// SIMATIC STEP 7 (V5.x) project Lit_servis
// CPU: CPU 312
// station: Hardware
// station: SIMATIC 300(1)
// station: P_ADR_BUS
// station: P_ADR_BUS
// station: Configuration
// program: S7 Program(6)

SYMBOL_TABLE
"s3.1-3.3"	I 4.0	BOOL	// авар. откл.ГП
"s3.4"	I 4.1	BOOL	// откл. вентилятора.
"s3.5"	I 4.2	BOOL	// вкл. вентилятора
"s3.6"	I 4.3	BOOL	// нормальное откл.ГП
"s3.7"	I 4.4	BOOL	// вкл. ГП
"s4.1"	I 4.5	BOOL	// выбор режима
"s4.2"	I 4.6	BOOL	// не используется в ПрП
"s4.3"	I 4.7	BOOL	// не используется в ПрП
"s1.1-1.2"	I 5.0	BOOL	// конеч. пол. левого 1
"s1.3-1.4"	I 5.1	BOOL	// конеч. пол. правого 1
"s1.5-1.6"	I 5.2	BOOL	// конеч. пол. левого 2
"s1.7-1.8"	I 5.3	BOOL	// конеч. пол. правого 2
"s1.9-1.10"	I 5.4	BOOL	// поднятие магазина
"s1.11"	I 5.5	BOOL	// положение штурвала
"s1.12"	I 5.6	BOOL	// контроль вентилятора
"B1.1"	I 5.7	BOOL	// наличие воздуха
"F1.1-1.3"	I 6.0	BOOL	// тепловое реле
"B8.1"	I 6.1	BOOL	// наличие крышки-левая
"B8.2"	I 6.2	BOOL	// сектор-левая
"B8.3"	I 6.3	BOOL	// наличие крышки-правая
"B8.4"	I 6.4	BOOL	// сектор-правая
"B8.5"	I 6.5	BOOL	// счётчик-левая
"B8.6"	I 6.6	BOOL	// счётчик-правая
"B8.7"	I 6.7	BOOL	// мёртвая точка
"B8.9"	I 7.0	BOOL	// min. магазин 1-левый
"B8.10"	I 7.1	BOOL	// max. магазин 1-левый
"B8.11"	I 7.2	BOOL	// min. магазин 2-правый
"B8.12"	I 7.3	BOOL	// max. магазин 2-правый
"K9.1"	Q 10.0	BOOL	// управление вентилятором
"K9.3"	Q 10.1	BOOL	// управление осн. нагревателем
"K9.4"	Q 10.2	BOOL	// управление 1 доп.. нагревателем
"K9.5"	Q 10.3	BOOL	// управление 2 доп.. нагревателем
"K9.6"	Q 10.4	BOOL	// управление-маг. колесо
"K9.7"	Q 10.5	BOOL	// управление-привод гумир.
"K1.12"	Q 10.6	BOOL	// управление-привод ГП
"K7.5"	Q 11.0	BOOL	// управление подачей крышек-магазин 1(левый)
"K7.10"	Q 11.1	BOOL	// управление подачей крышек-магазин 2(правый)
"K7.6"	Q 11.2	BOOL	// управление-грибок магазин 1(левый)
"K7.11"	Q 11.3	BOOL	// управление-грибок магазин 2(правый)
"Y2.1"	Q 11.4	BOOL	// подача пасты-левый
"Y2.2"	Q 11.5	BOOL	// подача пасты-правый
"Y2.9"	Q 11.6	BOOL	// управление тормозом
"VAT_1"	VAT 1	
END_SYMBOL_TABLE

FUNCTION FC 1 : VOID
VERSION : 0.1
BEGIN
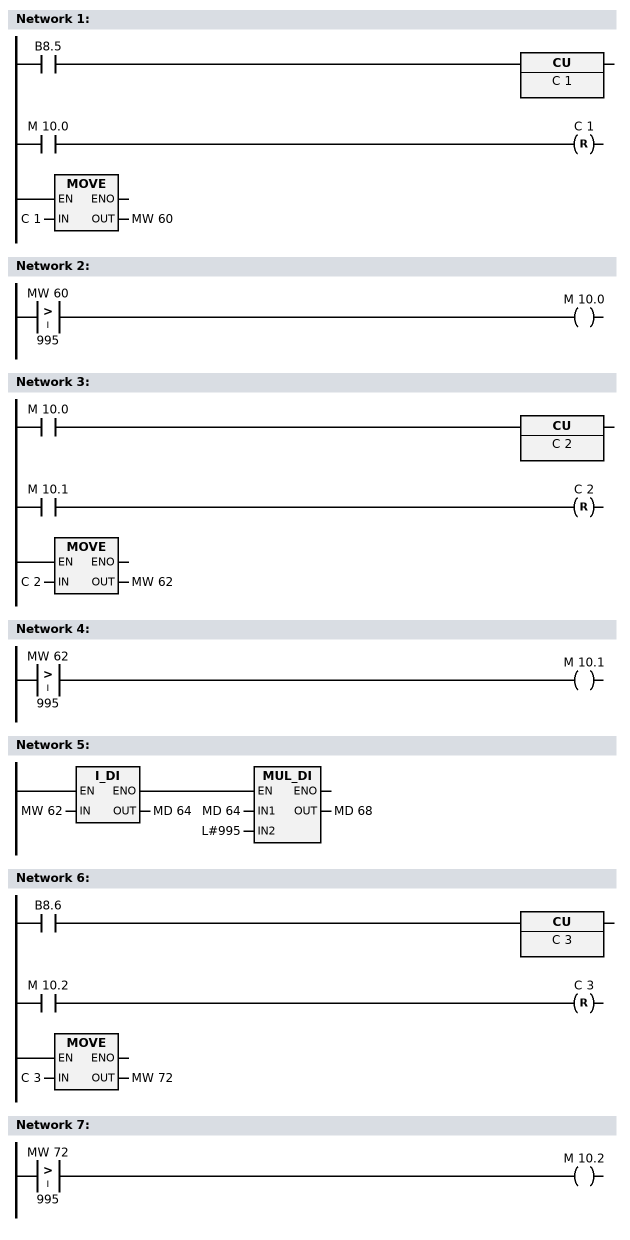
NETWORK
TITLE =
      A     "B8.5";
      CU    C 1;
      BLD   101;
      NOP   0;
      NOP   0;
      A     M 10.0;
      R     C 1;
      L     C 1;
      T     MW 60;
      NOP   0;
      NOP   0;
NETWORK
TITLE =
      L     MW 60;
      L     995;
      >I;
      =     M 10.0;
NETWORK
TITLE =
      A     M 10.0;
      CU    C 2;
      BLD   101;
      NOP   0;
      NOP   0;
      A     M 10.1;
      R     C 2;
      L     C 2;
      T     MW 62;
      NOP   0;
      NOP   0;
NETWORK
TITLE =
      L     MW 62;
      L     995;
      >I;
      =     M 10.1;
NETWORK
TITLE =
      A(;
      L     MW 62;
      ITD;
      T     MD 64;
      SET;
      SAVE;
      CLR;
      A     BR;
      );
      JNB   _001;
      L     MD 64;
      L     L#995;
      *D;
      T     MD 68;
_001: NOP   0;
NETWORK
TITLE =
      A     "B8.6";
      CU    C 3;
      BLD   101;
      NOP   0;
      NOP   0;
      A     M 10.2;
      R     C 3;
      L     C 3;
      T     MW 72;
      NOP   0;
      NOP   0;
NETWORK
TITLE =
      L     MW 72;
      L     995;
      >I;
      =     M 10.2;
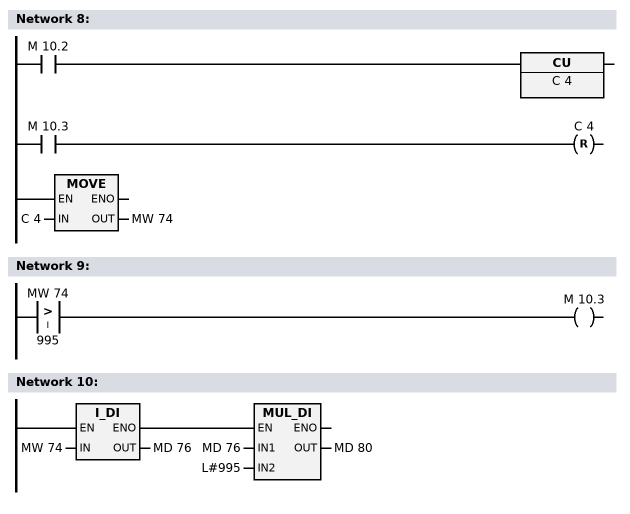
NETWORK
TITLE =
      A     M 10.2;
      CU    C 4;
      BLD   101;
      NOP   0;
      NOP   0;
      A     M 10.3;
      R     C 4;
      L     C 4;
      T     MW 74;
      NOP   0;
      NOP   0;
NETWORK
TITLE =
      L     MW 74;
      L     995;
      >I;
      =     M 10.3;
NETWORK
TITLE =
      A(;
      L     MW 74;
      ITD;
      T     MD 76;
      SET;
      SAVE;
      CLR;
      A     BR;
      );
      JNB   _002;
      L     MD 76;
      L     L#995;
      *D;
      T     MD 80;
_002: NOP   0;
NETWORK
TITLE =
END_FUNCTION

FUNCTION FC 2 : VOID
//Счётчики
VERSION : 0.1
BEGIN
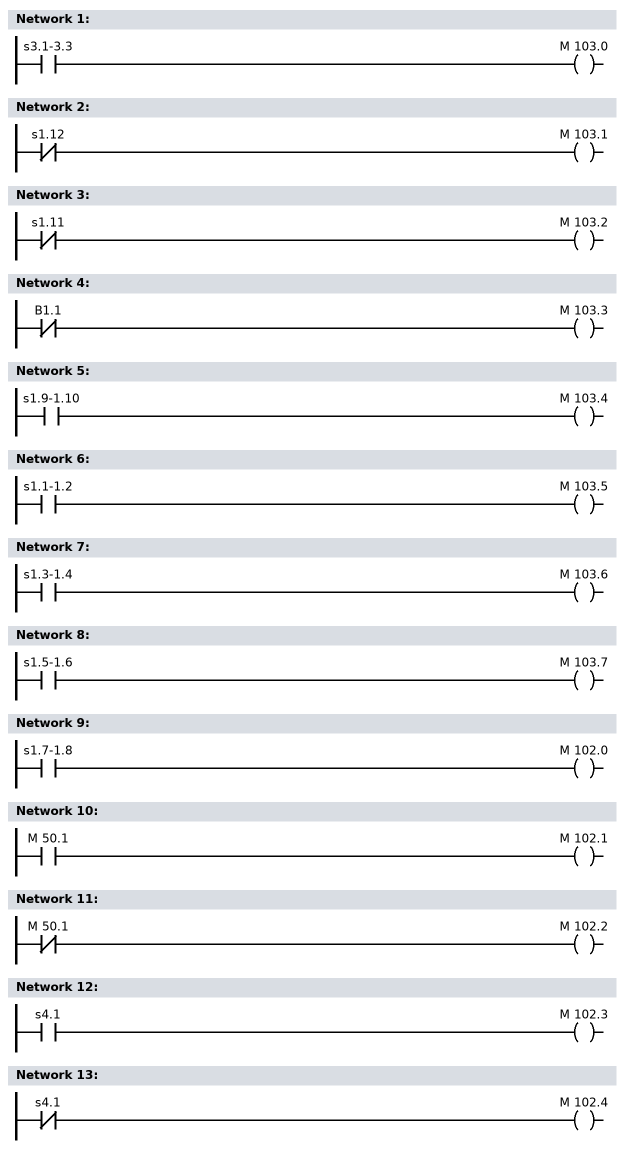
NETWORK
TITLE =
//Сообщение:аврийное отключение ГП
      A     "s3.1-3.3";
      =     M 103.0;
NETWORK
TITLE =
//Сообщение:вентилятор отключился
      AN    "s1.12";
      =     M 103.1;
NETWORK
TITLE =
//Сообщение:штурвал не в "автомате"
      AN    "s1.11";
      =     M 103.2;
NETWORK
TITLE =
//Сообщение:отсутствует воздух в системе
      AN    "B1.1";
      =     M 103.3;
NETWORK
TITLE =
//Сообщение:гумировочная головка магазин крышек подняты
      A     "s1.9-1.10";
      =     M 103.4;
NETWORK
TITLE =
//Сообщение:конечное положение левого 1 шнека
      A     "s1.1-1.2";
      =     M 103.5;
NETWORK
TITLE =
//Сообщение:конечное положение правого 1 шнека
      A     "s1.3-1.4";
      =     M 103.6;
NETWORK
TITLE =
//Сообщение:конечное положение левого 2 шнека
      A     "s1.5-1.6";
      =     M 103.7;
NETWORK
TITLE =
//Сообщение:конечное положение правого 2 шнека
      A     "s1.7-1.8";
      =     M 102.0;
NETWORK
TITLE =
//Сообщение:температура в норме
      A     M 50.1;
      =     M 102.1;
NETWORK
TITLE =
//Сообщение:температура ниже нормы
      AN    M 50.1;
      =     M 102.2;
NETWORK
TITLE =
//Сообщение:работа в автоматическом режиме
      A     "s4.1";
      =     M 102.3;
NETWORK
TITLE =
//Сообщение:работа в ручном режиме
      AN    "s4.1";
      =     M 102.4;
END_FUNCTION

ORGANIZATION_BLOCK OB 1
TITLE = "Main Program Sweep (Cycle)"
VERSION : 0.1
VAR_TEMP
  OB1_EV_CLASS : BYTE ;	//Bits 0-3 = 1 (Coming event), Bits 4-7 = 1 (Event class 1)
  OB1_SCAN_1 : BYTE ;	//1 (Cold restart scan 1 of OB 1), 3 (Scan 2-n of OB 1)
  OB1_PRIORITY : BYTE ;	//Priority of OB Execution
  OB1_OB_NUMBR : BYTE ;	//1 (Organization block 1, OB1)
  OB1_RESERVED_1 : BYTE ;	//Reserved for system
  OB1_RESERVED_2 : BYTE ;	//Reserved for system
  OB1_PREV_CYCLE : INT ;	//Cycle time of previous OB1 scan (milliseconds)
  OB1_MIN_CYCLE : INT ;	//Minimum cycle time of OB1 (milliseconds)
  OB1_MAX_CYCLE : INT ;	//Maximum cycle time of OB1 (milliseconds)
  OB1_DATE_TIME : DATE_AND_TIME ;	//Date and time OB1 started
END_VAR
BEGIN
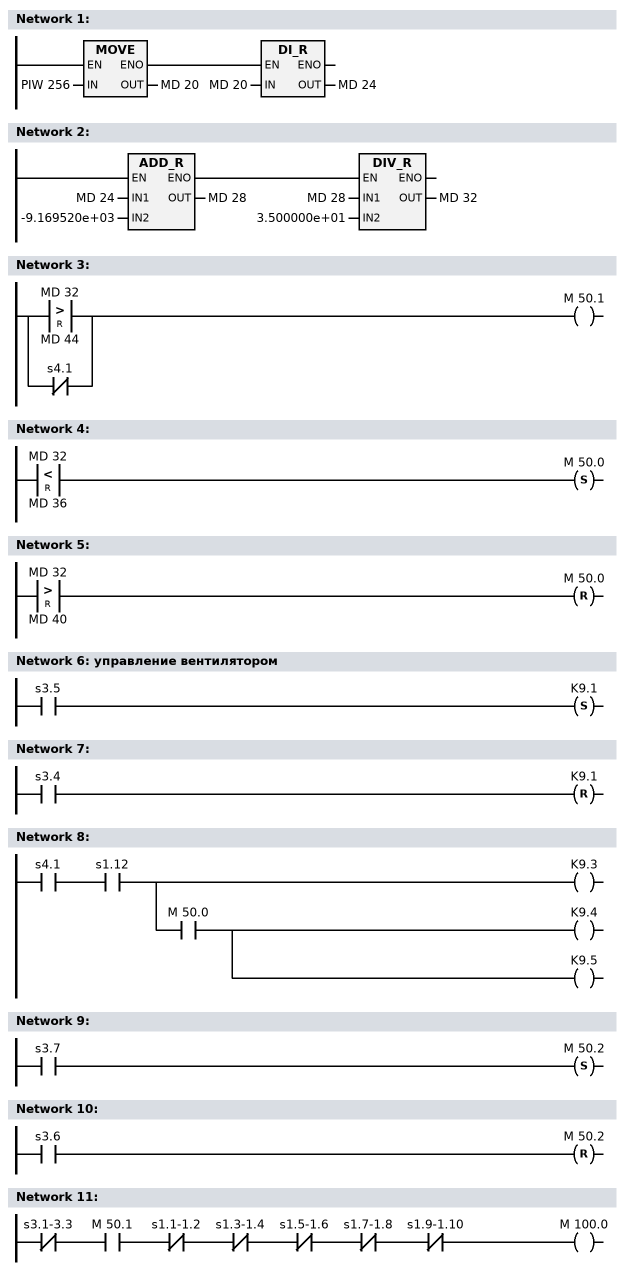
NETWORK
TITLE =
//измерение температуры
      A(;
      L     PIW 256;
      T     MD 20;
      SET;
      SAVE;
      CLR;
      A     BR;
      );
      JNB   _001;
      L     MD 20;
      DTR;
      T     MD 24;
_001: NOP   0;
NETWORK
TITLE =
//измерение температуры
      A(;
      L     MD 24;
      L     -9.169520e+03;
      +R;
      T     MD 28;
      AN    OV;
      SAVE;
      CLR;
      A     BR;
      );
      JNB   _002;
      L     MD 28;
      L     3.500000e+01;
      /R;
      T     MD 32;
_002: NOP   0;
NETWORK
TITLE =
//подготовка вкл. ГП либо при t=MD44 в авт.режиме, либо напрямую в ручном режиме 
      O(;
      L     MD 32;
      L     MD 44;
      >R;
      );
      ON    "s4.1";
      =     M 50.1;
NETWORK
TITLE =
//вкл. доп. нагревателей
      L     MD 32;
      L     MD 36;
      <R;
      S     M 50.0;
NETWORK
TITLE =
//откл. доп. нагревателей
      L     MD 32;
      L     MD 40;
      >R;
      R     M 50.0;
NETWORK
TITLE = управление вентилятором
//вкл. вентилятора
      A     "s3.5";
      S     "K9.1";
NETWORK
TITLE =
//откл. вентилятора
      A     "s3.4";
      R     "K9.1";
NETWORK
TITLE =
//вкл. основной нагреватель
      A     "s4.1";
      A     "s1.12";
      =     L 20.0;
      A     L 20.0;
      BLD   102;
      =     "K9.3";
      A     L 20.0;
      A     M 50.0;
      =     "K9.4";
      =     "K9.5";
NETWORK
TITLE =
//вкл. ГП кнопкой "пуск" на пульте
      A     "s3.7";
      S     M 50.2;
NETWORK
TITLE =
//откл. ГП кнопкой "стоп" на пульте
      A     "s3.6";
      R     M 50.2;
NETWORK
TITLE =
//вкл. и откл. ГП, магнитного колеса и привода гумирования
      AN    "s3.1-3.3";
      A     M 50.1;
      AN    "s1.1-1.2";
      AN    "s1.3-1.4";
      AN    "s1.5-1.6";
      AN    "s1.7-1.8";
      AN    "s1.9-1.10";
      =     M 100.0;
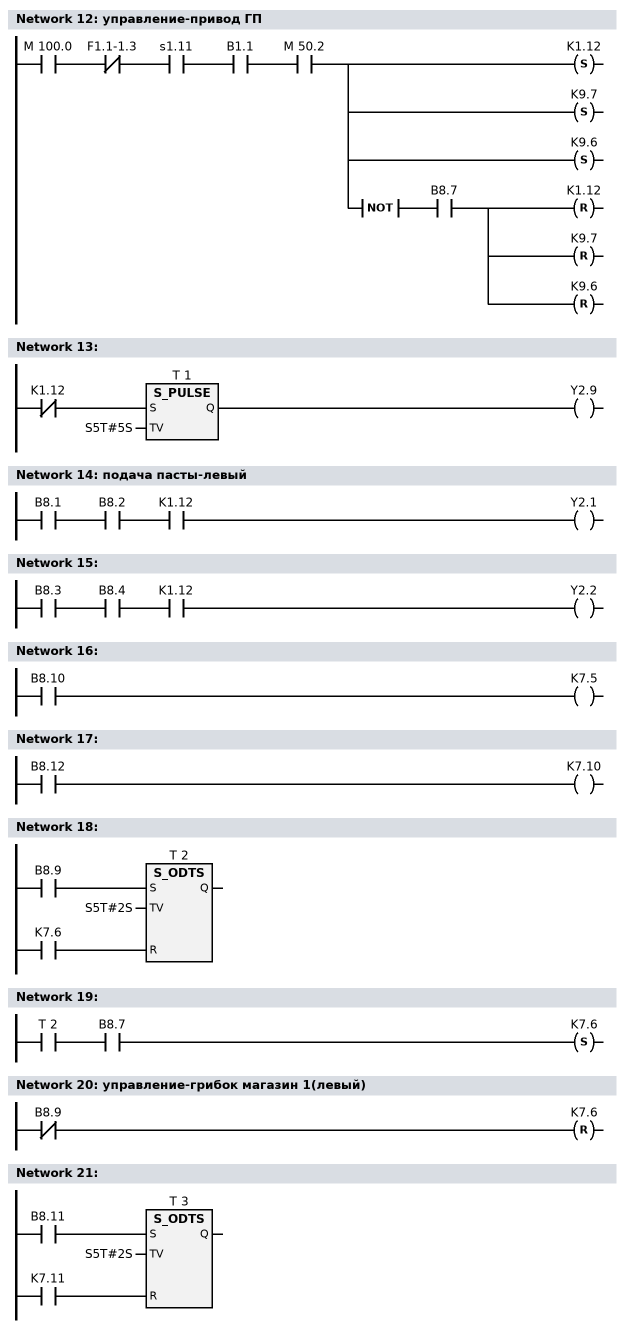
NETWORK
TITLE = управление-привод ГП
//вкл. и откл. ГП, магнитного колеса и привода гумирования (продолжение цепи)
      A     M 100.0;
      AN    "F1.1-1.3";
      A     "s1.11";
      A     "B1.1";
      A     M 50.2;
      =     L 20.0;
      A     L 20.0;
      BLD   102;
      S     "K1.12";
      A     L 20.0;
      BLD   102;
      S     "K9.7";
      A     L 20.0;
      BLD   102;
      S     "K9.6";
      A     L 20.0;
      NOT;
      A     "B8.7";
      R     "K1.12";
      R     "K9.7";
      R     "K9.6";
NETWORK
TITLE =
//откл. тормоз
      AN    "K1.12";
      L     S5T#5S;
      SP    T 1;
      NOP   0;
      NOP   0;
      NOP   0;
      A     T 1;
      =     "Y2.9";
NETWORK
TITLE = подача пасты-левый
//вкл. подачу пасты- левая крышка
      A     "B8.1";
      A     "B8.2";
      A     "K1.12";
      =     "Y2.1";
NETWORK
TITLE =
//вкл. подачу пасты- правая крышка
      A     "B8.3";
      A     "B8.4";
      A     "K1.12";
      =     "Y2.2";
NETWORK
TITLE =
//блокировка подачи крышек в левый магазин по "max"
      A     "B8.10";
      =     "K7.5";
NETWORK
TITLE =
//блокировка подачи крышек в правый магазин по "max"
      A     "B8.12";
      =     "K7.10";
NETWORK
TITLE =
//выдержка времени при появлении сигнала "min"-левый магазин
      A     "B8.9";
      L     S5T#2S;
      SS    T 2;
      A     "K7.6";
      R     T 2;
      NOP   0;
      NOP   0;
      NOP   0;
NETWORK
TITLE =
//блокировка поднятия крышки-левый магазин
      A     T 2;
      A     "B8.7";
      S     "K7.6";
NETWORK
TITLE = управление-грибок магазин 1(левый)
//снятие блокировки поднятия крышки-левый магазин
      AN    "B8.9";
      R     "K7.6";
NETWORK
TITLE =
//выдержка времени при появлении сигнала "min"-правый магазин
      A     "B8.11";
      L     S5T#2S;
      SS    T 3;
      A     "K7.11";
      R     T 3;
      NOP   0;
      NOP   0;
      NOP   0;
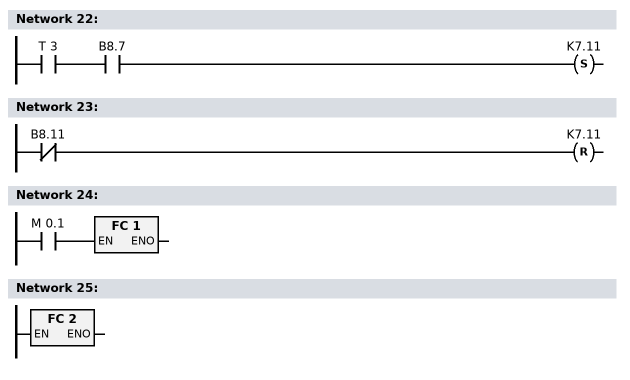
NETWORK
TITLE =
//блокировка поднятия крышки-правый магазин
      A     T 3;
      A     "B8.7";
      S     "K7.11";
NETWORK
TITLE =
//снятие блокировки поднятия крышки-правый магазин
      AN    "B8.11";
      R     "K7.11";
NETWORK
TITLE =
//вызов функции счёта крышек
      A     M 0.1;
      JNB   _003;
      CALL  FC 1;
_003: NOP   0;
NETWORK
TITLE =
//вызов функции формирования сообщений на ТP 177А
      CALL  FC 2;
      NOP   0;
END_ORGANIZATION_BLOCK
